PROGRAM P_Demo_Int64Add64
VAR
    liAccum : T_LARGE_INTEGER;; // 累计差值
    liDelta : T_LARGE_INTEGER;; // 本次差值
    bAdd    : BOOL;
END_VAR

// ============================================================
// Tc2_Utilities.Int64Add64 演示程序（FUNCTION，单周期触发）
// ============================================================
// 场景：累计差值（可正可负）求合，确认不会超 2⁶³ 后用本函数。
// 价值：替代手写有符号双倍长加；一行调用。
// 验证步骤：
//   1. 把本 PROGRAM 加到 PlcTask 调用列表
//   2. 编译 + 登录
//   3. 在线把 b... 触发位置 TRUE 一个周期
//   4. 观察输出变量是否符合期望
// ============================================================

IF bAdd THEN
    liAccum := Int64Add64(liAccum, liDelta);
    bAdd := FALSE;
END_IF;

END_PROGRAM

(* stored: Version 1.1.0.1, ProductVersion 3.1.4024.5
   POU P_Demo_Int64Add64: Id {0421705e-37af-5a57-94c0-aba067d581d7}, SpecialFunc None *)
